(* IEC 61131-3 sources: SafePLC-Gen-Evaluation/Evaluation Results/butane/run_02, 2 files *)

(* ---- io_declarations.st ---- *)
(* ==================================================  *)
(* PLC I/O Variable Declarations — CODESYS 3.5  *)
(* Generated by SafePLC-Gen Multimodal  *)
(* ==================================================  *)

VAR_GLOBAL
    (* --- Analog Inputs ---  *)
    TI_2909_Raw                  AT %IW0       : INT := 0;    (* TI-2909 — Temperature indicator on inlet piping to  *)
    TI_2917HH_Raw                AT %IW2       : INT := 0;    (* TI-2917HH — Temperature indicator high-high alarm, s  *)
    TT_2909_Raw                  AT %IW4       : INT := 0;    (* TT-2909 — Temperature transmitter on inlet line to  *)
    TT_2911_Raw                  AT %IW6       : INT := 0;    (* TT-2911 — Temperature transmitter on outlet line f  *)
    TT_2917_Raw                  AT %IW8       : INT := 0;    (* TT-2917 — Temperature transmitter on outlet/downst  *)
    XI_2901A_Raw                 AT %IW10      : INT := 0;    (* XI-2901A — Status indicator AVAILABLE for pump A, p  *)
    XI_2901B_Raw                 AT %IW12      : INT := 0;    (* XI-2901B — Status indicator AVAILABLE for pump B, p  *)
    (* --- Analog Outputs ---  *)
    HY_2903A_Out                 AT %QW0       : INT := 0;    (* HY-2903A — Hand relay/solenoid or I/P converter for  *)
    HY_2903B_Out                 AT %QW2       : INT := 0;    (* HY-2903B — Hand relay/solenoid or I/P converter for  *)
    KV_2904_Out                  AT %QW4       : INT := 0;    (* KV-2904 — Control valve KV-2904 on inlet utility/b  *)
    (* --- Digital Inputs ---  *)
    HS_2901A                     AT %IX0.0     : BOOL := FALSE;    (* HS-2901A — Hand switch for pump A (NOTE 9), manual   *)
    HS_2901A1                    AT %IX0.1     : BOOL := FALSE;    (* HS-2901A1 — Hand switch LOCAL/REMOTE selector for pu  *)
    HS_2901A2                    AT %IX0.2     : BOOL := FALSE;    (* HS-2901A2 — Hand switch STOP/START for pump A at MCC  *)
    HS_2901B                     AT %IX0.3     : BOOL := FALSE;    (* HS-2901B — Hand switch for pump B (NOTE 9), manual   *)
    HS_2901B1                    AT %IX0.4     : BOOL := FALSE;    (* HS-2901B1 — Hand switch LOCAL/REMOTE selector for pu  *)
    HS_2901B2                    AT %IX0.5     : BOOL := FALSE;    (* HS-2901B2 — Hand switch STOP/START for pump B at MCC  *)
    HS_EMERGENCY_STOP_A_2901A    AT %IX0.6     : BOOL := FALSE;    (* HS-EMERGENCY-STOP-A-2901A — Hand switch EMERGENCY STOP for pump A, l  *)
    HS_EMERGENCY_STOP_B_2901B    AT %IX0.7     : BOOL := FALSE;    (* HS-EMERGENCY-STOP-B-2901B — Hand switch EMERGENCY STOP for pump B, l  *)
    HS_START_STOP_A_2901A        AT %IX1.0     : BOOL := FALSE;    (* HS-START-STOP-A-2901A — Hand switch START/STOP for pump A, local  *)
    HS_START_STOP_B_2901B        AT %IX1.1     : BOOL := FALSE;    (* HS-START-STOP-B-2901B — Hand switch START/STOP for pump B, local  *)
    VSHH_2901A                   AT %IX1.2     : BOOL := FALSE;    (* VSHH-2901A — Vibration switch high-high on pump/motor  *)
    VSHH_2901B                   AT %IX1.3     : BOOL := FALSE;    (* VSHH-2901B — Vibration switch high-high on pump/motor  *)
    (* --- Digital Outputs ---  *)
    ESD_3200                     AT %QX0.0     : BOOL := FALSE;    (* ESD-3200 — Emergency shutdown system logic node, pa  *)
    MCC_2901A                    AT %QX0.1     : BOOL := FALSE;    (* MCC-2901A — Motor control centre / motor-operated co  *)
    MCC_2901B                    AT %QX0.2     : BOOL := FALSE;    (* MCC-2901B — Motor control centre / motor-operated co  *)
    PSD_2917                     AT %QX0.3     : BOOL := FALSE;    (* PSD-2917 — Pressure/temperature shutdown device ass  *)
    XV_RS_001A_BOT               AT %QX0.4     : BOOL := FALSE;    (* XV-RS-001A-BOT — RS isolation valve on bottom inlet nozzl  *)
    XV_RS_001A_TOP               AT %QX0.5     : BOOL := FALSE;    (* XV-RS-001A-TOP — RS (ring seal / spectacle blind or isola  *)
    XV_RS_001B_BOT               AT %QX0.6     : BOOL := FALSE;    (* XV-RS-001B-BOT — RS isolation valve on bottom outlet nozz  *)
    XV_RS_001B_TOP               AT %QX0.7     : BOOL := FALSE;    (* XV-RS-001B-TOP — RS isolation valve on top outlet nozzle   *)
END_VAR

(* ---- generated_code.st ---- *)
(* Generated by SafePLC-Gen Multimodal — CODESYS 3.5 *)
(* IEC 61131-3 Structured Text *)
(* Date: 2026-04-25T12:06:57.520952 *)

PROGRAM PumpStation_2901

VAR
    TI_2909_Raw                  AT %IW0       : INT := 0;
    TI_2917HH_Raw                AT %IW2       : INT := 0;
    TT_2909_Raw                  AT %IW4       : INT := 0;
    TT_2911_Raw                  AT %IW6       : INT := 0;
    TT_2917_Raw                  AT %IW8       : INT := 0;
    XI_2901A_Raw                 AT %IW10      : INT := 0;
    XI_2901B_Raw                 AT %IW12      : INT := 0;
    HY_2903A_Out                 AT %QW0       : INT := 0;
    HY_2903B_Out                 AT %QW2       : INT := 0;
    KV_2904_Out                  AT %QW4       : INT := 0;
    HS_2901A                     AT %IX0.0     : BOOL := FALSE;
    HS_2901A1                    AT %IX0.1     : BOOL := FALSE;
    HS_2901A2                    AT %IX0.2     : BOOL := FALSE;
    HS_2901B                     AT %IX0.3     : BOOL := FALSE;
    HS_2901B1                    AT %IX0.4     : BOOL := FALSE;
    HS_2901B2                    AT %IX0.5     : BOOL := FALSE;
    HS_EMERGENCY_STOP_A_2901A    AT %IX0.6     : BOOL := FALSE;
    HS_EMERGENCY_STOP_B_2901B    AT %IX0.7     : BOOL := FALSE;
    HS_START_STOP_A_2901A        AT %IX1.0     : BOOL := FALSE;
    HS_START_STOP_B_2901B        AT %IX1.1     : BOOL := FALSE;
    VSHH_2901A                   AT %IX1.2     : BOOL := FALSE;
    VSHH_2901B                   AT %IX1.3     : BOOL := FALSE;
    ESD_3200                     AT %QX0.0     : BOOL := FALSE;
    MCC_2901A                    AT %QX0.1     : BOOL := FALSE;
    MCC_2901B                    AT %QX0.2     : BOOL := FALSE;
    PSD_2917                     AT %QX0.3     : BOOL := FALSE;
    XV_RS_001A_BOT               AT %QX0.4     : BOOL := FALSE;
    XV_RS_001A_TOP               AT %QX0.5     : BOOL := FALSE;
    XV_RS_001B_BOT               AT %QX0.6     : BOOL := FALSE;
    XV_RS_001B_TOP               AT %QX0.7     : BOOL := FALSE;
END_VAR

VAR
    ESTOP                        : BOOL := FALSE;
    MANUAL_RESET                 : BOOL := FALSE;
    LOOP_2917_TRIP               : BOOL := FALSE;
    LOOP_2901A_TRIP              : BOOL := FALSE;
    LOOP_2901B_TRIP              : BOOL := FALSE;
    TT_2917_HH                   : BOOL := FALSE;
    TT_2917_LL                   : BOOL := FALSE;
    VSHH_2901A_HH                : BOOL := FALSE;
    VSHH_2901A_LL                : BOOL := FALSE;
    VSHH_2901B_HH                : BOOL := FALSE;
    VSHH_2901B_LL                : BOOL := FALSE;
    SAFE_STATE                   : BOOL := FALSE;
    FirstScan                    : BOOL := TRUE;

    TI_2909_Scaled               : REAL := 0.0;
    TI_2917HH_Scaled             : REAL := 0.0;
    TT_2909_Scaled               : REAL := 0.0;
    TT_2911_Scaled               : REAL := 0.0;
    TT_2917_Scaled               : REAL := 0.0;
    XI_2901A_Scaled              : REAL := 0.0;
    XI_2901B_Scaled              : REAL := 0.0;

    TI_2909_HH_SP                : REAL := 120.0;
    TI_2909_H_SP                 : REAL := 110.0;
    TI_2909_L_SP                 : REAL := 10.0;
    TI_2909_LL_SP                : REAL := 5.0;
    TI_2909_Deadband             : REAL := 2.0;
    TI_2909_H                    : BOOL := FALSE;
    TI_2909_L                    : BOOL := FALSE;
    TI_2909_HH_Latch             : SR := (S1 := FALSE, R := FALSE, Q1 := FALSE);
    TI_2909_LL_Latch             : SR := (S1 := FALSE, R := FALSE, Q1 := FALSE);
    TI_2909_HH_Ack               : BOOL := FALSE;
    TI_2909_LL_Ack               : BOOL := FALSE;

    TT_2909_HH_SP                : REAL := 120.0;
    TT_2909_H_SP                 : REAL := 110.0;
    TT_2909_L_SP                 : REAL := 10.0;
    TT_2909_LL_SP                : REAL := 5.0;
    TT_2909_Deadband             : REAL := 2.0;
    TT_2909_H                    : BOOL := FALSE;
    TT_2909_L                    : BOOL := FALSE;
    TT_2909_HH_Latch             : SR := (S1 := FALSE, R := FALSE, Q1 := FALSE);
    TT_2909_LL_Latch             : SR := (S1 := FALSE, R := FALSE, Q1 := FALSE);
    TT_2909_HH_Ack               : BOOL := FALSE;
    TT_2909_LL_Ack               : BOOL := FALSE;

    TT_2911_HH_SP                : REAL := 130.0;
    TT_2911_H_SP                 : REAL := 120.0;
    TT_2911_L_SP                 : REAL := 10.0;
    TT_2911_LL_SP                : REAL := 5.0;
    TT_2911_Deadband             : REAL := 2.0;
    TT_2911_H                    : BOOL := FALSE;
    TT_2911_L                    : BOOL := FALSE;
    TT_2911_HH_Latch             : SR := (S1 := FALSE, R := FALSE, Q1 := FALSE);
    TT_2911_LL_Latch             : SR := (S1 := FALSE, R := FALSE, Q1 := FALSE);
    TT_2911_HH_Ack               : BOOL := FALSE;
    TT_2911_LL_Ack               : BOOL := FALSE;

    TT_2917_HH_SP                : REAL := 140.0;
    TT_2917_H_SP                 : REAL := 130.0;
    TT_2917_L_SP                 : REAL := 10.0;
    TT_2917_LL_SP                : REAL := 5.0;
    TT_2917_Deadband             : REAL := 2.0;
    TT_2917_H                    : BOOL := FALSE;
    TT_2917_L                    : BOOL := FALSE;
    TT_2917_HH_Latch             : SR := (S1 := FALSE, R := FALSE, Q1 := FALSE);
    TT_2917_LL_Latch             : SR := (S1 := FALSE, R := FALSE, Q1 := FALSE);
    TT_2917_HH_Ack               : BOOL := FALSE;
    TT_2917_LL_Ack               : BOOL := FALSE;

    TI_2917HH_HH_SP              : REAL := 145.0;
    TI_2917HH_H_SP               : REAL := 135.0;
    TI_2917HH_L_SP               : REAL := 10.0;
    TI_2917HH_LL_SP              : REAL := 5.0;
    TI_2917HH_Deadband           : REAL := 2.0;
    TI_2917HH_H                  : BOOL := FALSE;
    TI_2917HH_L                  : BOOL := FALSE;
    TI_2917HH_HH_Latch           : SR := (S1 := FALSE, R := FALSE, Q1 := FALSE);
    TI_2917HH_LL_Latch           : SR := (S1 := FALSE, R := FALSE, Q1 := FALSE);
    TI_2917HH_HH_Ack             : BOOL := FALSE;
    TI_2917HH_LL_Ack             : BOOL := FALSE;

    XI_2901A_HH_SP               : REAL := 95.0;
    XI_2901A_H_SP                : REAL := 90.0;
    XI_2901A_L_SP                : REAL := 10.0;
    XI_2901A_LL_SP               : REAL := 5.0;
    XI_2901A_Deadband            : REAL := 2.0;
    XI_2901A_H                   : BOOL := FALSE;
    XI_2901A_L                   : BOOL := FALSE;
    XI_2901A_HH_Latch            : SR := (S1 := FALSE, R := FALSE, Q1 := FALSE);
    XI_2901A_LL_Latch            : SR := (S1 := FALSE, R := FALSE, Q1 := FALSE);
    XI_2901A_HH_Ack              : BOOL := FALSE;
    XI_2901A_LL_Ack              : BOOL := FALSE;

    XI_2901B_HH_SP               : REAL := 95.0;
    XI_2901B_H_SP                : REAL := 90.0;
    XI_2901B_L_SP                : REAL := 10.0;
    XI_2901B_LL_SP               : REAL := 5.0;
    XI_2901B_Deadband            : REAL := 2.0;
    XI_2901B_H                   : BOOL := FALSE;
    XI_2901B_L                   : BOOL := FALSE;
    XI_2901B_HH_Latch            : SR := (S1 := FALSE, R := FALSE, Q1 := FALSE);
    XI_2901B_LL_Latch            : SR := (S1 := FALSE, R := FALSE, Q1 := FALSE);
    XI_2901B_HH_Ack              : BOOL := FALSE;
    XI_2901B_LL_Ack              : BOOL := FALSE;

    KV_2904_SP                   : REAL := 80.0;
    KV_2904_Kp                   : REAL := 1.5;
    KV_2904_Ki                   : REAL := 0.05;
    KV_2904_Integral             : REAL := 0.0;
    KV_2904_Error                : REAL := 0.0;
    KV_2904_Output_Pct           : REAL := 0.0;

    HY_2903A_SP                  : REAL := 70.0;
    HY_2903A_Kp                  : REAL := 1.2;
    HY_2903A_Ki                  : REAL := 0.04;
    HY_2903A_Integral            : REAL := 0.0;
    HY_2903A_Error               : REAL := 0.0;
    HY_2903A_Output_Pct          : REAL := 0.0;

    HY_2903B_SP                  : REAL := 70.0;
    HY_2903B_Kp                  : REAL := 1.2;
    HY_2903B_Ki                  : REAL := 0.04;
    HY_2903B_Integral            : REAL := 0.0;
    HY_2903B_Error               : REAL := 0.0;
    HY_2903B_Output_Pct          : REAL := 0.0;

    PumpA_Run                    : BOOL := FALSE;
    PumpA_StartCmd               : BOOL := FALSE;
    PumpA_StopCmd                : BOOL := FALSE;
    PumpA_LatchS                 : BOOL := FALSE;
    PumpA_LatchR                 : BOOL := FALSE;

    PumpB_Run                    : BOOL := FALSE;
    PumpB_StartCmd               : BOOL := FALSE;
    PumpB_StopCmd                : BOOL := FALSE;
    PumpB_LatchS                 : BOOL := FALSE;
    PumpB_LatchR                 : BOOL := FALSE;

    XV_Enable_A                  : BOOL := FALSE;
    XV_Enable_B                  : BOOL := FALSE;

    System_Alarm                 : BOOL := FALSE;
END_VAR

IF FirstScan THEN
    LOOP_2917_TRIP  := TRUE;
    LOOP_2901A_TRIP := TRUE;
    LOOP_2901B_TRIP := TRUE;
    SAFE_STATE      := TRUE;
    MCC_2901A       := FALSE;
    MCC_2901B       := FALSE;
    PSD_2917        := FALSE;
    ESD_3200        := FALSE;
    XV_RS_001A_TOP  := FALSE;
    XV_RS_001A_BOT  := FALSE;
    XV_RS_001B_TOP  := FALSE;
    XV_RS_001B_BOT  := FALSE;
    HY_2903A_Out    := 6554;
    HY_2903B_Out    := 6554;
    KV_2904_Out     := 6554;
    PumpA_Run       := FALSE;
    PumpB_Run       := FALSE;
    FirstScan       := FALSE;
    RETURN;
END_IF;

ESTOP := HS_EMERGENCY_STOP_A_2901A OR HS_EMERGENCY_STOP_B_2901B;

TI_2909_Scaled   := ((INT_TO_REAL(TI_2909_Raw)   - 6554.0) / (32767.0 - 6554.0)) * 150.0;
TI_2917HH_Scaled := ((INT_TO_REAL(TI_2917HH_Raw) - 6554.0) / (32767.0 - 6554.0)) * 150.0;
TT_2909_Scaled   := ((INT_TO_REAL(TT_2909_Raw)   - 6554.0) / (32767.0 - 6554.0)) * 150.0;
TT_2911_Scaled   := ((INT_TO_REAL(TT_2911_Raw)   - 6554.0) / (32767.0 - 6554.0)) * 150.0;
TT_2917_Scaled   := ((INT_TO_REAL(TT_2917_Raw)   - 6554.0) / (32767.0 - 6554.0)) * 150.0;
XI_2901A_Scaled  := ((INT_TO_REAL(XI_2901A_Raw)  - 6554.0) / (32767.0 - 6554.0)) * 100.0;
XI_2901B_Scaled  := ((INT_TO_REAL(XI_2901B_Raw)  - 6554.0) / (32767.0 - 6554.0)) * 100.0;

TT_2917_HH    := TT_2917_Scaled > TT_2917_HH_SP;
TT_2917_LL    := TT_2917_Scaled < TT_2917_LL_SP;
VSHH_2901A_HH := VSHH_2901A;
VSHH_2901A_LL := FALSE;
VSHH_2901B_HH := VSHH_2901B;
VSHH_2901B_LL := FALSE;

IF TT_2917_HH OR TT_2917_LL THEN
    LOOP_2917_TRIP := TRUE;
ELSIF LOOP_2917_TRIP AND MANUAL_RESET AND NOT TT_2917_HH AND NOT TT_2917_LL THEN
    LOOP_2917_TRIP := FALSE;
END_IF;

IF VSHH_2901A_HH OR VSHH_2901A_LL THEN
    LOOP_2901A_TRIP := TRUE;
ELSIF LOOP_2901A_TRIP AND MANUAL_RESET AND NOT VSHH_2901A_HH AND NOT VSHH_2901A_LL THEN
    LOOP_2901A_TRIP := FALSE;
END_IF;

IF VSHH_2901B_HH OR VSHH_2901B_LL THEN
    LOOP_2901B_TRIP := TRUE;
ELSIF LOOP_2901B_TRIP AND MANUAL_RESET AND NOT VSHH_2901B_HH AND NOT VSHH_2901B_LL THEN
    LOOP_2901B_TRIP := FALSE;
END_IF;

SAFE_STATE := ESTOP OR LOOP_2917_TRIP OR LOOP_2901A_TRIP OR LOOP_2901B_TRIP;

ESD_3200 := NOT SAFE_STATE;
PSD_2917 := NOT LOOP_2917_TRIP;

TI_2909_HH_Latch(S1 := TI_2909_Scaled > TI_2909_HH_SP,
                 R  := TI_2909_HH_Ack AND (TI_2909_Scaled <= (TI_2909_HH_SP - TI_2909_Deadband)));
IF TI_2909_Scaled > TI_2909_H_SP THEN
    TI_2909_H := TRUE;
ELSIF TI_2909_Scaled <= (TI_2909_H_SP - TI_2909_Deadband) THEN
    TI_2909_H := FALSE;
END_IF;
IF TI_2909_Scaled < TI_2909_L_SP THEN
    TI_2909_L := TRUE;
ELSIF TI_2909_Scaled >= (TI_2909_L_SP + TI_2909_Deadband) THEN
    TI_2909_L := FALSE;
END_IF;
TI_2909_LL_Latch(S1 := TI_2909_Scaled < TI_2909_LL_SP,
                 R  := TI_2909_LL_Ack AND (TI_2909_Scaled >= (TI_2909_LL_SP + TI_2909_Deadband)));

TT_2909_HH_Latch(S1 := TT_2909_Scaled > TT_2909_HH_SP,
                 R  := TT_2909_HH_Ack AND (TT_2909_Scaled <= (TT_2909_HH_SP - TT_2909_Deadband)));
IF TT_2909_Scaled > TT_2909_H_SP THEN
    TT_2909_H := TRUE;
ELSIF TT_2909_Scaled <= (TT_2909_H_SP - TT_2909_Deadband) THEN
    TT_2909_H := FALSE;
END_IF;
IF TT_2909_Scaled < TT_2909_L_SP THEN
    TT_2909_L := TRUE;
ELSIF TT_2909_Scaled >= (TT_2909_L_SP + TT_2909_Deadband) THEN
    TT_2909_L := FALSE;
END_IF;
TT_2909_LL_Latch(S1 := TT_2909_Scaled < TT_2909_LL_SP,
                 R  := TT_2909_LL_Ack AND (TT_2909_Scaled >= (TT_2909_LL_SP + TT_2909_Deadband)));

TT_2911_HH_Latch(S1 := TT_2911_Scaled > TT_2911_HH_SP,
                 R  := TT_2911_HH_Ack AND (TT_2911_Scaled <= (TT_2911_HH_SP - TT_2911_Deadband)));
IF TT_2911_Scaled > TT_2911_H_SP THEN
    TT_2911_H := TRUE;
ELSIF TT_2911_Scaled <= (TT_2911_H_SP - TT_2911_Deadband) THEN
    TT_2911_H := FALSE;
END_IF;
IF TT_2911_Scaled < TT_2911_L_SP THEN
    TT_2911_L := TRUE;
ELSIF TT_2911_Scaled >= (TT_2911_L_SP + TT_2911_Deadband) THEN
    TT_2911_L := FALSE;
END_IF;
TT_2911_LL_Latch(S1 := TT_2911_Scaled < TT_2911_LL_SP,
                 R  := TT_2911_LL_Ack AND (TT_2911_Scaled >= (TT_2911_LL_SP + TT_2911_Deadband)));

TT_2917_HH_Latch(S1 := TT_2917_Scaled > TT_2917_HH_SP,
                 R  := TT_2917_HH_Ack AND (TT_2917_Scaled <= (TT_2917_HH_SP - TT_2917_Deadband)));
IF TT_2917_Scaled > TT_2917_H_SP THEN
    TT_2917_H := TRUE;
ELSIF TT_2917_Scaled <= (TT_2917_H_SP - TT_2917_Deadband) THEN
    TT_2917_H := FALSE;
END_IF;
IF TT_2917_Scaled < TT_2917_L_SP THEN
    TT_2917_L := TRUE;
ELSIF TT_2917_Scaled >= (TT_2917_L_SP + TT_2917_Deadband) THEN
    TT_2917_L := FALSE;
END_IF;
TT_2917_LL_Latch(S1 := TT_2917_Scaled < TT_2917_LL_SP,
                 R  := TT_2917_LL_Ack AND (TT_2917_Scaled >= (TT_2917_LL_SP + TT_2917_Deadband)));

TI_2917HH_HH_Latch(S1 := TI_2917HH_Scaled > TI_2917HH_HH_SP,
                   R  := TI_2917HH_HH_Ack AND (TI_2917HH_Scaled <= (TI_2917HH_HH_SP - TI_2917HH_Deadband)));
IF TI_2917HH_Scaled > TI_2917HH_H_SP THEN
    TI_2917HH_H := TRUE;
ELSIF TI_2917HH_Scaled <= (TI_2917HH_H_SP - TI_2917HH_Deadband) THEN
    TI_2917HH_H := FALSE;
END_IF;
IF TI_2917HH_Scaled < TI_2917HH_L_SP THEN
    TI_2917HH_L := TRUE;
ELSIF TI_2917HH_Scaled >= (TI_2917HH_L_SP + TI_2917HH_Deadband) THEN
    TI_2917HH_L := FALSE;
END_IF;
TI_2917HH_LL_Latch(S1 := TI_2917HH_Scaled < TI_2917HH_LL_SP,
                   R  := TI_2917HH_LL_Ack AND (TI_2917HH_Scaled >= (TI_2917HH_LL_SP + TI_2917HH_Deadband)));

XI_2901A_HH_Latch(S1 := XI_2901A_Scaled > XI_2901A_HH_SP,
                  R  := XI_2901A_HH_Ack AND (XI_2901A_Scaled <= (XI_2901A_HH_SP - XI_2901A_Deadband)));
IF XI_2901A_Scaled > XI_2901A_H_SP THEN
    XI_2901A_H := TRUE;
ELSIF XI_2901A_Scaled <= (XI_2901A_H_SP - XI_2901A_Deadband) THEN
    XI_2901A_H := FALSE;
END_IF;
IF XI_2901A_Scaled < XI_2901A_L_SP THEN
    XI_2901A_L := TRUE;
ELSIF XI_2901A_Scaled >= (XI_2901A_L_SP + XI_2901A_Deadband) THEN
    XI_2901A_L := FALSE;
END_IF;
XI_2901A_LL_Latch(S1 := XI_2901A_Scaled < XI_2901A_LL_SP,
                  R  := XI_2901A_LL_Ack AND (XI_2901A_Scaled >= (XI_2901A_LL_SP + XI_2901A_Deadband)));

XI_2901B_HH_Latch(S1 := XI_2901B_Scaled > XI_2901B_HH_SP,
                  R  := XI_2901B_HH_Ack AND (XI_2901B_Scaled <= (XI_2901B_HH_SP - XI_2901B_Deadband)));
IF XI_2901B_Scaled > XI_2901B_H_SP THEN
    XI_2901B_H := TRUE;
ELSIF XI_2901B_Scaled <= (XI_2901B_H_SP - XI_2901B_Deadband) THEN
    XI_2901B_H := FALSE;
END_IF;
IF XI_2901B_Scaled < XI_2901B_L_SP THEN
    XI_2901B_L := TRUE;
ELSIF XI_2901B_Scaled >= (XI_2901B_L_SP + XI_2901B_Deadband) THEN
    XI_2901B_L := FALSE;
END_IF;
XI_2901B_LL_Latch(S1 := XI_2901B_Scaled < XI_2901B_LL_SP,
                  R  := XI_2901B_LL_Ack AND (XI_2901B_Scaled >= (XI_2901B_LL_SP + XI_2901B_Deadband)));

PumpA_StartCmd := (HS_2901A OR HS_START_STOP_A_2901A) AND NOT SAFE_STATE;
PumpA_StopCmd  := SAFE_STATE OR HS_2901A2;
PumpA_LatchS   := PumpA_StartCmd AND NOT PumpA_StopCmd;
PumpA_LatchR   := PumpA_StopCmd;
IF PumpA_LatchS THEN
    PumpA_Run := TRUE;
ELSIF PumpA_LatchR THEN
    PumpA_Run := FALSE;
END_IF;

PumpB_StartCmd := (HS_2901B OR HS_START_STOP_B_2901B) AND NOT SAFE_STATE;
PumpB_StopCmd  := SAFE_STATE OR HS_2901B2;
PumpB_LatchS   := PumpB_StartCmd AND NOT PumpB_StopCmd;
PumpB_LatchR   := PumpB_StopCmd;
IF PumpB_LatchS THEN
    PumpB_Run := TRUE;
ELSIF PumpB_LatchR THEN
    PumpB_Run := FALSE;
END_IF;

XV_Enable_A := PumpA_Run AND NOT SAFE_STATE;
XV_Enable_B := PumpB_Run AND NOT SAFE_STATE;

XV_RS_001A_TOP := XV_Enable_A;
XV_RS_001A_BOT := XV_Enable_A;
XV_RS_001B_TOP := XV_Enable_B;
XV_RS_001B_BOT := XV_Enable_B;

IF NOT SAFE_STATE THEN
    MCC_2901A := PumpA_Run AND (HS_2901A1 OR HS_2901A);
    MCC_2901B := PumpB_Run AND (HS_2901B1 OR HS_2901B);

    HY_2903A_Error    := HY_2903A_SP - TT_2909_Scaled;
    HY_2903A_Integral := HY_2903A_Integral + (HY_2903A_Ki * HY_2903A_Error);
    IF HY_2903A_Integral > 100.0 THEN
        HY_2903A_Integral := 100.0;
    ELSIF HY_2903A_Integral < 0.0 THEN
        HY_2903A_Integral := 0.0;
    END_IF;
    HY_2903A_Output_Pct := (HY_2903A_Kp * HY_2903A_Error) + HY_2903A_Integral;
    IF HY_2903A_Output_Pct > 100.0 THEN
        HY_2903A_Output_Pct := 100.0;
    ELSIF HY_2903A_Output_Pct < 0.0 THEN
        HY_2903A_Output_Pct := 0.0;
    END_IF;
    HY_2903A_Out := REAL_TO_INT(6554.0 + (HY_2903A_Output_Pct / 100.0) * (32767.0 - 6554.0));

    HY_2903B_Error    := HY_2903B_SP - TT_2917_Scaled;
    HY_2903B_Integral := HY_2903B_Integral + (HY_2903B_Ki * HY_2903B_Error);
    IF HY_2903B_Integral > 100.0 THEN
        HY_2903B_Integral := 100.0;
    ELSIF HY_2903B_Integral < 0.0 THEN
        HY_2903B_Integral := 0.0;
    END_IF;
    HY_2903B_Output_Pct := (HY_2903B_Kp * HY_2903B_Error) + HY_2903B_Integral;
    IF HY_2903B_Output_Pct > 100.0 THEN
        HY_2903B_Output_Pct := 100.0;
    ELSIF HY_2903B_Output_Pct < 0.0 THEN
        HY_2903B_Output_Pct := 0.0;
    END_IF;
    HY_2903B_Out := REAL_TO_INT(6554.0 + (HY_2903B_Output_Pct / 100.0) * (32767.0 - 6554.0));

    KV_2904_Error    := KV_2904_SP - TT_2911_Scaled;
    KV_2904_Integral := KV_2904_Integral + (KV_2904_Ki * KV_2904_Error);
    IF KV_2904_Integral > 100.0 THEN
        KV_2904_Integral := 100.0;
    ELSIF KV_2904_Integral < 0.0 THEN
        KV_2904_Integral := 0.0;
    END_IF;
    KV_2904_Output_Pct := (KV_2904_Kp * KV_2904_Error) + KV_2904_Integral;
    IF KV_2904_Output_Pct > 100.0 THEN
        KV_2904_Output_Pct := 100.0;
    ELSIF KV_2904_Output_Pct < 0.0 THEN
        KV_2904_Output_Pct := 0.0;
    END_IF;
    KV_2904_Out := REAL_TO_INT(6554.0 + (KV_2904_Output_Pct / 100.0) * (32767.0 - 6554.0));
ELSE
    MCC_2901A    := FALSE;
    MCC_2901B    := FALSE;
    HY_2903A_Out := 6554;
    HY_2903B_Out := 6554;
    KV_2904_Out  := 6554;
END_IF;

System_Alarm :=
    TI_2909_HH_Latch.Q1   OR TI_2909_LL_Latch.Q1   OR TI_2909_H   OR TI_2909_L   OR
    TT_2909_HH_Latch.Q1   OR TT_2909_LL_Latch.Q1   OR TT_2909_H   OR TT_2909_L   OR
    TT_2911_HH_Latch.Q1   OR TT_2911_LL_Latch.Q1   OR TT_2911_H   OR TT_2911_L   OR
    TT_2917_HH_Latch.Q1   OR TT_2917_LL_Latch.Q1   OR TT_2917_H   OR TT_2917_L   OR
    TI_2917HH_HH_Latch.Q1 OR TI_2917HH_LL_Latch.Q1 OR TI_2917HH_H OR TI_2917HH_L OR
    XI_2901A_HH_Latch.Q1  OR XI_2901A_LL_Latch.Q1  OR XI_2901A_H  OR XI_2901A_L  OR
    XI_2901B_HH_Latch.Q1  OR XI_2901B_LL_Latch.Q1  OR XI_2901B_H  OR XI_2901B_L  OR
    LOOP_2917_TRIP OR LOOP_2901A_TRIP OR LOOP_2901B_TRIP OR SAFE_STATE;

END_PROGRAM
